// TIA Portal V19 export
VAR_GLOBAL   // PLC tag table "A01_SensorMatPresence"
   S1_MaterialPresence_Straightener_Entry AT %I26.7 : Bool;   // CC1 506SQ1 / 736BF2
   S2_MaterialPresence_Straightener_Exit AT %I29.6 : Bool;   // CC1 506SQ2 / 837BF1
   S3_MaterialPresence_JBPinchRoll_Exit AT %I29.7 : Bool;   // CC1 557SQ2 / 837BF2
END_VAR
